FUNCTION_BLOCK FB_DCMotor
VAR_INPUT
END_VAR

VAR_OUTPUT
END_VAR

VAR
	_Alarm												: BOOL;
	fb_DebugCart_AP240Power								: DFB_Cylinder;
	fb_DebugCart_Col_PCWValve							: DFB_Cylinder;
	
	_AP240Power_Perm									: WORD;
	_AP240Power_SD										: WORD;
	_Col_PCWValve_Perm									: WORD;
	_Col_PCWValve_SD									: WORD;
	
	_DUT_DebugCart_AP240Power							: DUT_Cylinder;
	_DUT_DebugCart_Col_PCWValve							: DUT_Cylinder;
END_VAR

/////////////////////////////////////////////////////////////////////////////////////////////////////////////////////////////////////////////////////////////////////////////////
//	
/////////////////////////////////////////////////////////////////////////////////////////////////////////////////////////////////////////////////////////////////////////////////

(*
IF DewPoint_Abort OR OFA6Bar_Abort THEN
	_Alarm		:= TRUE;
ELSIF (NOT ALM_DCCOL.AlarmID[E_DCFACAlarm.eCriticalCondensationAlarm]) AND (NOT ALM_DCCOL.AlarmID[E_DCFACAlarm.e6BarLowOFAAirPressureAlarm]) THEN
	_Alarm		:= FALSE;
END_IF

_DUT_DebugCart_AP240Power.AutInp		:= DebugCart_APPresentSignal AND (NOT FluidLeakageSignal) AND (NOT GroundFault) AND (NOT _Alarm);
											//(NOT DewPoint_Abort) AND 
											//(NOT OFA6Bar_Abort) AND (NOT ALM_DCCOL.AlarmID[E_DCFACAlarm.e6BarLowOFAAirPressureAlarm]) AND 
											//(NOT ALM_DCCOL.AlarmID[E_DCFACAlarm.eCriticalCondensationAlarm]);

fb_DebugCart_AP240Power(
	Sec_P		:= Sec_P, 
	ID		:= 'DebugCart AP240Power', 
	Simulate		:= _DUT_DebugCart_AP240Power.Simulate, 
	Permissive		:= _AP240Power_Perm, 
	ShutDown		:= _AP240Power_SD, 
	AutoInp		:= _DUT_DebugCart_AP240Power.AutInp, 
	Command		:= _DUT_DebugCart_AP240Power.CMD, 
	IExtend		:= DebugCart_APPowerOnSignal, 
	IRetract		:= (NOT DebugCart_APPowerOnSignal), 
	Travel_Time		:= _DUT_DebugCart_AP240Power.Travel_Time, 
	SetOutput_Pulse		:= FALSE, 
	FailedHoldLast		:= FALSE,
	OExtend		=> DebugCart_APPowerOn, 
	ORetract		=> , 
	DUT		:= _DUT_DebugCart_AP240Power);

*)


	
PermSD();





_DUT_DebugCart_Col_PCWValve.AutInp		:= (NOT ALM_DCCOL.AlarmID[E_DCFACAlarm.eSystemPCWLeakageAlarm]) AND
											(NOT ALM_DCCOL.AlarmID[E_DCFACAlarm.eSystemPCWSupplyLeakageAlarm]) AND
											(NOT ALM_DCCOL.AlarmID[E_DCFACAlarm.eSystemPCWReturnLeakageAlarm]) AND
											(NOT ALM_DCCOL.AlarmID[E_DCFACAlarm.eCriticalCondensationAlarm]) AND 
											(NOT ALM_DCCOL.AlarmID[E_DCFACAlarm.e6BarLowOFAAirPressureAlarm])AND 
											(NOT DewPoint_Abort) AND
											(NOT OFA6Bar_Abort);

					
fb_DebugCart_Col_PCWValve(
	Sec_P:= Sec_P, 
	ID:= 'DebugCart Column PCW Valve', 
	Simulate:= _DUT_DebugCart_Col_PCWValve.Simulate, 
	Permissive:= _Col_PCWValve_Perm,  //check before execute
	ShutDown:= _Col_PCWValve_SD,  //keep checking this condition 
	AutoInp:= _DUT_DebugCart_Col_PCWValve.AutInp, 
	Command:= _DUT_DebugCart_Col_PCWValve.CMD, //1: Retract, 2: Extend, 4: Auto
	IExtend:= DebugCart_ColumnPCWValve, 
	IRetract:= (NOT DebugCart_ColumnPCWValve), 
	Travel_Time:= _DUT_DebugCart_Col_PCWValve.Travel_Time, //detect input after output trigger
	SetOutput_Pulse:= FALSE,  //output rising edge
	FailedHoldLast:= FALSE,  //remain state after failed. 1: Remain, 0: FALSE
	OExtend=> DebugCart_ColumnPCWValve,  //map to output variable
	ORetract=> , 
	DUT:= _DUT_DebugCart_Col_PCWValve);

ACTION PermSD:
FC_BitToWord(
	BOOL_00		:= TRUE, 
	BOOL_01		:= TRUE, 
	BOOL_02		:= TRUE, 
	BOOL_03		:= TRUE, 
	BOOL_04		:= TRUE, 
	BOOL_05		:= TRUE, 
	BOOL_06		:= TRUE, 
	BOOL_07		:= TRUE, 
	BOOL_08		:= TRUE, 
	BOOL_09		:= TRUE, 
	BOOL_10		:= TRUE, 
	BOOL_11		:= TRUE, 
	BOOL_12		:= TRUE, 
	BOOL_13		:= TRUE, 
	BOOL_14		:= TRUE, 
	BOOL_15		:= TRUE, 
	Output_Word		=> _Col_PCWValve_Perm);
	
FC_BitToWord(
	BOOL_00		:= FALSE, 
	BOOL_01		:= FALSE, 
	BOOL_02		:= FALSE, 
	BOOL_03		:= FALSE, 
	BOOL_04		:= FALSE, 
	BOOL_05		:= FALSE, 
	BOOL_06		:= FALSE, 
	BOOL_07		:= FALSE, 
	BOOL_08		:= FALSE, 
	BOOL_09		:= FALSE, 
	BOOL_10		:= FALSE, 
	BOOL_11		:= FALSE, 
	BOOL_12		:= FALSE, 
	BOOL_13		:= FALSE, 
	BOOL_14		:= FALSE, 
	BOOL_15		:= FALSE, 
	Output_Word		=> _Col_PCWValve_SD);
END_ACTION

END_FUNCTION_BLOCK

(* stored: Version 1.1.0.1, ProductVersion 3.1.4022.18
   POU FB_DCMotor: Id {c17387f9-d74e-48e2-9e05-34b020aa612c}, SpecialFunc None
   Action PermSD: Id {f9871df8-4830-4d77-a1c4-fe839ea41fec} *)
